{attribute 'qualified_only'}
VAR_GLOBAL
		
	bEmergencyButton 	: BOOL;

	bEnableU 			: BOOL;
	bEnableFF 			: BOOL;
	bEnablePID 			: BOOL;
	bEnableFlowShare	: BOOL;
	
	bEnableOne			: BOOL;
	bEnableTwo			: BOOL;
	bEnableThree		: BOOL;	
	
	bHoldButton 		: BOOL;
	
	bErrorOne 			: BOOL;
	bErrorTwo			: BOOL;
	bErrorThree			: BOOL;
	
	bSineMotion			: BOOL;
	bRampMotion			: BOOL;
	bRampAxis			: BOOL;
	bHoming				: BOOL;
	
	// Modes
	bAuto				: BOOL;
	bManual				: BOOL;
	bManDirect			: BOOL;
	bManConst			: BOOL;
	bManSpeed			: BOOL;
	
	// Config Enables
	bConfigJoysticks	: BOOL;
END_VAR

(* stored: Version 1.1.0.1
   GVL G_Enables: Id {0aed01c2-6407-4abd-87cb-b561ebe6419c} *)
